PROGRAM D_Regul_Humi
VAR
	TON_Humi: TON;
	TOF_Deshu: TOF;

	Cons_Regul_Humi: REAL;
	Cons_Regul_Deshu: REAL;
	Interdiction_Humi: BOOL;
	Interdiction_Deshu: BOOL;
	Bool_Reg_Humi: BOOL;
	Bool_Reg_Deshu: BOOL;
	
	Regul_humidification: OSCAT_BASIC.CTRL_PID;
	Sup_PID_humi: REAL := 0;
	Regul_Deshumidification: OSCAT_BASIC.CTRL_PID;
	Sup_PID_Deshu: REAL := 0;
	SCL_Real_Humi: SCL_Real;
	SCL_Real_Deshu: SCL_Real;
	Dew_Point_Mes: Dew_Point;
	Dew_Point_Cons: Dew_Point;
	Mesure_Dew_Point: REAL;
	Consigne_Dew_Point: REAL;
	RS_Deshu: RS;
	RS_enable: RS;
END_VAR
VAR // added by the converter: edge detectors and wires of the graphical bodies
    _w1, _w3, _w4 : ANY;
    _w2 : BOOL;
END_VAR

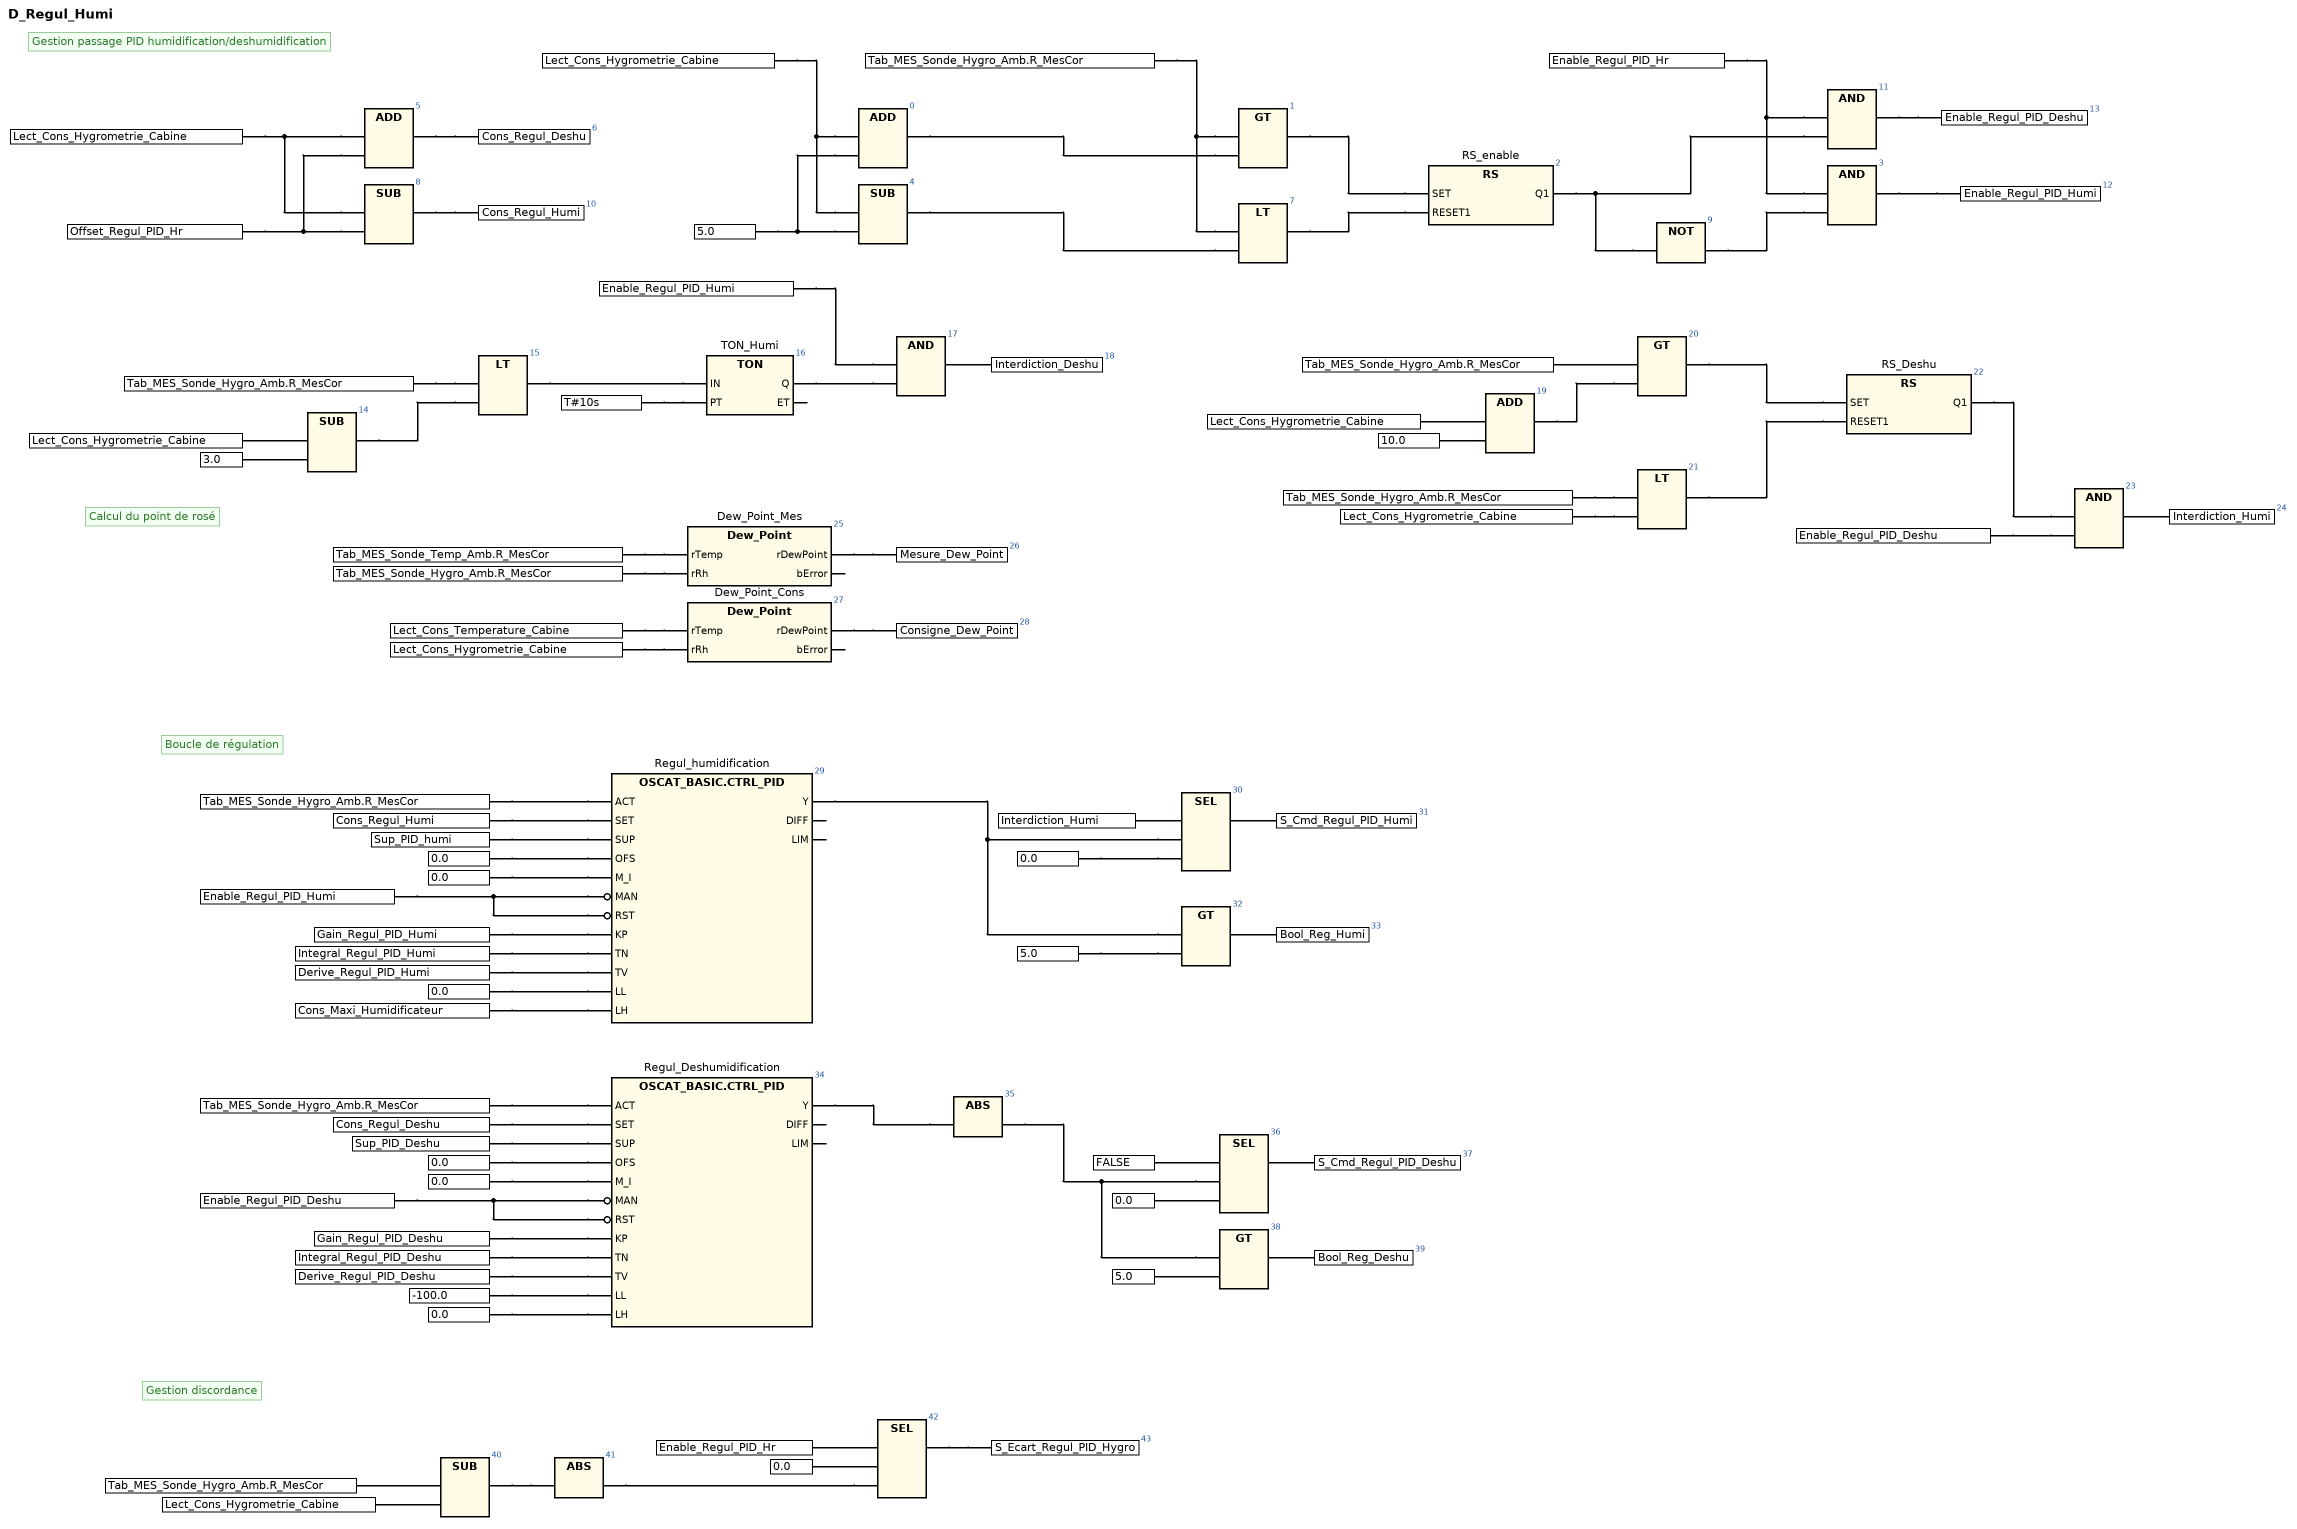
RS_enable(SET := Tab_MES_Sonde_Hygro_Amb.R_MesCor > Lect_Cons_Hygrometrie_Cabine + 5.0, RESET1 := _w1); // RS
_w3 := Enable_Regul_PID_Hr AND _w2;
// Gestion passage PID humidification/deshumidification
Cons_Regul_Deshu := Lect_Cons_Hygrometrie_Cabine + Offset_Regul_PID_Hr;
_w1 := Tab_MES_Sonde_Hygro_Amb.R_MesCor < Lect_Cons_Hygrometrie_Cabine - 5.0;
_w2 := NOT RS_enable.Q1;
Cons_Regul_Humi := Lect_Cons_Hygrometrie_Cabine - Offset_Regul_PID_Hr;
Enable_Regul_PID_Humi := _w3;
Enable_Regul_PID_Deshu := Enable_Regul_PID_Hr AND RS_enable.Q1;
TON_Humi(IN := Tab_MES_Sonde_Hygro_Amb.R_MesCor < Lect_Cons_Hygrometrie_Cabine - 3.0, PT := T#10s); // TON
Interdiction_Deshu := Enable_Regul_PID_Humi AND TON_Humi.Q;
RS_Deshu(SET := Tab_MES_Sonde_Hygro_Amb.R_MesCor > Lect_Cons_Hygrometrie_Cabine + 10.0, RESET1 := Tab_MES_Sonde_Hygro_Amb.R_MesCor < Lect_Cons_Hygrometrie_Cabine); // RS
Interdiction_Humi := RS_Deshu.Q1 AND Enable_Regul_PID_Deshu;
// Calcul du point de rosé
Dew_Point_Mes(rTemp := Tab_MES_Sonde_Temp_Amb.R_MesCor, rRh := Tab_MES_Sonde_Hygro_Amb.R_MesCor); // Dew_Point
Mesure_Dew_Point := Dew_Point_Mes.rDewPoint;
Dew_Point_Cons(rTemp := Lect_Cons_Temperature_Cabine, rRh := Lect_Cons_Hygrometrie_Cabine); // Dew_Point
Consigne_Dew_Point := Dew_Point_Cons.rDewPoint;
// Boucle de régulation
Regul_humidification(
    ACT := Tab_MES_Sonde_Hygro_Amb.R_MesCor,
    SET := Cons_Regul_Humi,
    SUP := Sup_PID_humi,
    OFS := 0.0,
    M_I := 0.0,
    MAN := NOT Enable_Regul_PID_Humi,
    RST := NOT Enable_Regul_PID_Humi,
    KP := Gain_Regul_PID_Humi,
    TN := Integral_Regul_PID_Humi,
    TV := Derive_Regul_PID_Humi,
    LL := 0.0,
    LH := Cons_Maxi_Humidificateur); // OSCAT_BASIC.CTRL_PID
S_Cmd_Regul_PID_Humi := SEL(Interdiction_Humi, Regul_humidification.Y, 0.0);
Bool_Reg_Humi := Regul_humidification.Y > 5.0;
Regul_Deshumidification(
    ACT := Tab_MES_Sonde_Hygro_Amb.R_MesCor,
    SET := Cons_Regul_Deshu,
    SUP := Sup_PID_Deshu,
    OFS := 0.0,
    M_I := 0.0,
    MAN := NOT Enable_Regul_PID_Deshu,
    RST := NOT Enable_Regul_PID_Deshu,
    KP := Gain_Regul_PID_Deshu,
    TN := Integral_Regul_PID_Deshu,
    TV := Derive_Regul_PID_Deshu,
    LL := -100.0,
    LH := 0.0); // OSCAT_BASIC.CTRL_PID
_w4 := ABS(Regul_Deshumidification.Y);
S_Cmd_Regul_PID_Deshu := SEL(FALSE, _w4, 0.0);
Bool_Reg_Deshu := _w4 > 5.0;
// Gestion discordance
S_Ecart_Regul_PID_Hygro := SEL(Enable_Regul_PID_Hr, 0.0, ABS(Tab_MES_Sonde_Hygro_Amb.R_MesCor - Lect_Cons_Hygrometrie_Cabine));

END_PROGRAM

(* stored: Version 1.1.0.1, ProductVersion 3.1.4024.16
   POU D_Regul_Humi: Id {4fcdaa42-c83a-4369-9b1c-0251747f304b}, SpecialFunc None *)
